PROGRAM MAIN
VAR
END_VAR

struct_text_ex();

END_PROGRAM

(* stored: Version 1.1.0.1, ProductVersion 3.1.4024.9
   POU MAIN: Id {8ffc1a15-8f1b-4a5b-a2c5-b2bfb9a41400}, SpecialFunc None *)
